# B&R Automation Studio project RobotNewEra
Automation Studio 4.2.4.149; 2.0.0

## Configuration APC820

CPU 5PC900.TS77-00, AutomationRuntime D4.21, Build 4.1.2, Safety 0.0

### Hardware
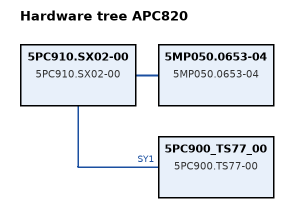
```
5MP050.0653-04 : 5MP050.0653-04 v1.0.3.0  [ETH1 -> 5PC910.SX02-00.IF3 (NodeNumber=1)]
  Terminal = true
  VncVcObjectName = Visu
  VncKeyMappingFile = VC\5MP050.0653-04.dis
  VncMaxConnections = 4
  VncRefreshRate = 100
5PC900_TS77_00 : 5PC900.TS77-00 v1.0.0.2  [SY -> 5PC910.SX02-00.SY1]
  UserRamDevice = APC8xx.SRAM
  UserRamSize = 770048
  RemMemDevice = APC8xx.SRAM
  RemMemSize = 261888
  PermanentPvSize = 10000
  RemanentGlobalPvSize = 81920
  VolatileGlobalPvSize = 500000
  PreservePermanentPvMemory = 1
  EnableUsbRemoteInstall = 1
  Connections = 8
  TimerDeviceType = EPLX2X
  TimerDevice = 5PC820.SX01-00.IF6
  TaskClassIdleTime = 8000
  Cyclic1Duration = 2000
  Cyclic1Tolerance = 0
  Cyclic1Stack = 40000
  Cyclic1Output = 1
  Cyclic2Duration = 30000
  Cyclic2Tolerance = 60000
  Cyclic2Stack = 28192
  Cyclic3Duration = 50000
  Cyclic3Tolerance = 200000
  Cyclic3Stack = 10240
  Cyclic4Duration = 100000
  Cyclic4Tolerance = 100000
  Cyclic5Duration = 200000
  Cyclic5Tolerance = 200000
  Cyclic6Duration = 500000
  Cyclic6Tolerance = 500000
  Cyclic7Duration = 1000000
  Cyclic7Tolerance = 1000000
  Cyclic8Duration = 30000
  Cyclic8Tolerance = 30000000
  Cyclic8Stack = 38192
5PC910.SX02-00 : 5PC910.SX02-00 v1.3.0.0
  Connector IF3:
    ActivateDevice = 1
    Mode = Manual
    InternetAddress = 192.168.1.9
    SubnetMask = 255.255.255.0
  Connector IF4:
    ActivateDevice = 1
    Mode = Manual
    SubnetMask = 255.255.255.0
```

### Cpu.per - 5PC900_TS77_00/Cpu.per
```iecst
(********************************************************************
 * COPYRIGHT --
 ********************************************************************
 * File: Cpu.per
 * Author: renj
 * Created: November 07, 2014
 ********************************************************************
 * Declaration of permanent variables
 ********************************************************************)
VAR_CONFIG
	HmiRetain AT %M0; (* *)
END_VAR
```

### AXESMap.ncm - 5PC900_TS77_00/Motion/AXESMap.ncm
```
NcMapping (NcSwId=ACP10)
  NcObject gAxisX (ModuleAddress=SDC_IF1.ST1, InterfaceType=SDC, Type=ncAXIS, Channel=1, AcoposSimulation=Off, InitParameter=sdc_i, AcoposParameter=sdc_p, AdditionalData=CNC_Enabled="1", Disabled=FALSE, ModuleDisabled=FALSE)
  NcObject gAxisY (ModuleAddress=SDC_IF1.ST2, InterfaceType=SDC, Type=ncAXIS, Channel=1, AcoposSimulation=Off, InitParameter=sdc_i, AcoposParameter=sdc_p, AdditionalData=CNC_Enabled="1", Disabled=FALSE)
  NcObject gAxisZ (ModuleAddress=SDC_IF1.ST3, InterfaceType=SDC, Type=ncAXIS, Channel=1, AcoposSimulation=Off, InitParameter=sdc_i, AcoposParameter=sdc_p, AdditionalData=CNC_Enabled="1", Disabled=FALSE)
  NcObject gAxisA (ModuleAddress=SDC_IF1.ST4, InterfaceType=SDC, Type=ncAXIS, Channel=1, AcoposSimulation=Off, InitParameter=sdc_i, AcoposParameter=sdc_p, AdditionalData=CNC_Enabled="1", Disabled=FALSE)
  NcObject gAxisB (ModuleAddress=SDC_IF1.ST5, InterfaceType=SDC, Type=ncAXIS, Channel=1, AcoposSimulation=Off, InitParameter=sdc_i, AcoposParameter=sdc_p, AdditionalData=CNC_Enabled="1", Disabled=FALSE)
  NcObject gAxisC (ModuleAddress=SDC_IF1.ST6, InterfaceType=SDC, Type=ncAXIS, Channel=1, AcoposSimulation=Off, InitParameter=sdc_i, AcoposParameter=sdc_p, AdditionalData=CNC_Enabled="1", Disabled=FALSE)
```

### Acp10cfg.ncc - 5PC900_TS77_00/Motion/Acp10cfg.ncc
```
NcConfiguration (Version=2.46.0, NcSwId=Acp10)
  ACP10CF1_typ:
    cnt_nettrc_rec_drive = 150
    bufsize_trace_upload = 1200
    tc_nc_man_task = Cyclic #1
    glob_pv_as_ncobject = Yes
    ncsys_dl_broadcast = Yes
    ncsys_dl_acp_reset = Yes
    safemc_log_err_to_ax = Yes
    network_init:
      ncsw_init_execute = Yes
      automatic_execute = No
      node_nr_warning = Yes
      net_err_before_ncact = Yes
    nettrc:
      enter_parsecrec = Yes
      enter_ncaction = Yes
      save_ring_startidx = No
    cam_prof_download:
      cam_dat_dl_parallel = No
      tc_cam_dl_parallel = Task class for NC Manager task
    plk_if[0]:
      if_name = IF6
      tc_CycDat_PLCopen = Task class for NC Manager task
      mc_broadcast_extdat = No
    sdc_if[0]:
      if_name = SDC_IF1
      mc_broadcast_size = 800
      mc_broadcast_extdat = No
```

### CNCMap.ncm - 5PC900_TS77_00/Motion/CNCMap.ncm
```
NcMapping (NcSwId=ARNC0)
  NcObject gRobot (Type=ncCNCSYS, Channel=1, AcoposSimulation=Off, InitParameter=cnc_i, Disabled=FALSE, ModuleDisabled=FALSE)
```

### MotionPvMa.vvm - 5PC900_TS77_00/Motion/MotionPvMa.vvm
```iecst
(********************************************************************
 * COPYRIGHT -- Bernecker + Rainer
 ********************************************************************
 * File: MotionPvMap.vvm
 * Author: radaka
 * Created: June 29, 2009
 ********************************************************************
 * PV mapping file
 ********************************************************************)
VAR_CONFIG
	Config.Config.Output.Monitor.ConfigOk AT %Q.Axes.Axes[0].Input.Parameter.ConfigOk; (*Insert your comment here...*)
	Config.Config.Output.Monitor.ConfigOk AT %Q.Cnc.Cnc[0].Input.Parameter.ConfigOk; (*Insert your comment here...*)
	Config.Config.Output.Monitor.ConfigOk AT %Q.System.System[0].Input.Parameter.ConfigOk; (*Insert your comment here...*)
	System.System[0].Output.Monitor.SystemAddress AT %Q.Config.Config.Input.Parameter.SystemAddress; (*Insert your comment here...*)
	Cnc.Cnc[0].Output.Monitor.CncAddress AT %Q.Config.Config.Input.Parameter.CncAddress; (*Insert your comment here...*)
	Axes.Axes[0].Output.Monitor.AxesAddress AT %Q.Config.Config.Input.Parameter.AxesAddress; (*Insert your comment here...*)
	Axes.Axes[0].Output.Monitor.AxesAddress AT %Q.System.System[0].Input.Parameter.AxesAddress; (*Insert your comment here...*)
	Cnc.Cnc[0].Output.Monitor.CncAddress AT %Q.System.System[0].Input.Parameter.CncAddress; (*Insert your comment here...*)
	Axes.Axes[0].Output.Monitor.AxesAddress AT %Q.Trf.AxesAddress; (*Only if TRF is used*)
	Cnc.Cnc[0].Output.Monitor.CncAddress AT %Q.Jog.CncAddress; (*Insert your comment here...*)
	Axes.Axes[0].Output.Monitor.AxesAddress AT %Q.6axATrqFF.AxesAddress; (*Insert your comment here...*)
END_VAR
```

## Configuration APC910

CPU 5PC900.TS77-02, AutomationRuntime N4.06, Build 4.1.2

### Task classes (Cpu.sw)
```

```

### Hardware
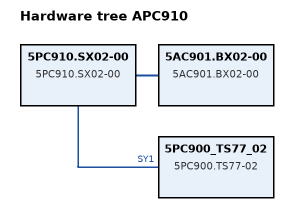
```
5AC901.BX02-00 : 5AC901.BX02-00 v1.0.0.2  [SY -> 5PC910.SX02-00.SY3]
5PC900_TS77_02 : 5PC900.TS77-02 v1.0.0.2  [SY -> 5PC910.SX02-00.SY1]
  Cyclic1Duration = 10000
  Cyclic1Tolerance = 10000
  Cyclic2Duration = 20000
  Cyclic2Tolerance = 20000
  Cyclic3Duration = 50000
  Cyclic3Tolerance = 50000
  Cyclic4Duration = 100000
  Cyclic4Tolerance = 100000
  Cyclic5Duration = 200000
  Cyclic5Tolerance = 200000
  Cyclic6Duration = 500000
  Cyclic6Tolerance = 500000
  Cyclic7Duration = 1000000
  Cyclic7Tolerance = 1000000
  Cyclic8Duration = 10000
  Cyclic8Tolerance = 30000000
5PC910.SX02-00 : 5PC910.SX02-00 v1.3.0.0
  Connector IF3:
    ActivateDevice = 1
    Mode = Manual
    InternetAddress = 192.168.0.9
    SubnetMask = 255.255.255.0
  Connector IF4:
    ActivateDevice = 1
    Mode = Manual
    InternetAddress = 192.168.1.9
    SubnetMask = 255.255.255.0
```

## Configuration Simulation

CPU , AutomationRuntime D4.24, Build 4.1.2, Safety 1.5

### Task classes (Cpu.sw)
```
Cyclic#1 (cycle 2000 us, tolerance 0 us):
  OptMotion <- MotionHandling.Optimizer.OptMotion.prg
  Cnc <- MotionHandling.CncHandling.Cnc.prg
  System <- MotionHandling.SystemHandling.System.prg (Version=1.00.1)
  Axes <- MotionHandling.AxesHandling.Axes.prg
  Jog <- MotionHandling.Jogging.Jog.prg
  Config <- MotionHandling.Configuration.Config.prg
  Trf <- MotionHandling.Transformations.Trf.prg
  myRecipe <- (binary)
Cyclic#2 (cycle 30000 us, tolerance 1200000 us):
  Error <- ErrorHandling.Error.prg  // Error Handling
  HmiKeyCtrl <- HmiHandling.HmiKeyCtrl.HmiKeyCtrl.prg
Cyclic#3 (cycle 20000 us, tolerance 10000000 us):
  HmiPrg <- HmiHandling.HmiPrg.HmiPrg.prg  // C++ Implementation FileExplorer
Cyclic#8 (cycle 30000 us, tolerance 30000000 us):
  HmiAlarm <- HmiHandling.HmiAlarm.HmiAlarm.prg
  HmiMain <- HmiHandling.HmiMain.HmiMain.prg
  HmiFile <- HmiHandling.HmiMain.HmiFile.prg
  HmiJogCtrl <- HmiHandling.HmiJog.HmiJogCtrl.prg
  RecipeCont <- Recipe.RecipeControl.prg
  UserStd <- UserStd.UserStd.prg  // User Management
  HmiHardKey <- HmiHandling.HmiHardKey.HmiHardKeyCtrl.prg  // HardKey Simulation
  HmiEditor <- HmiHandling.HmiEditor.HmiEditor.prg
  HmiFileVar <- HmiHandling.HmiEditor.HmiFileVar.prg
  HmiSetup <- HmiHandling.HmiSetup.HmiSetup.prg
NcDataObjects: sdc_p <- MotionHandling.MotionInitFiles.SDC.sdc_p.dob, ps_p <- MotionHandling.MotionInitFiles.ps_p.dob, sdc_i <- MotionHandling.MotionInitFiles.SDC.sdc_i.dob, AcpError <- MotionHandling.AxesHandling.AcpError.dob, sdc_j1_i <- MotionHandling.MotionInitFiles.SDC.sdc_j1_i.dob, sdc_j2_i <- MotionHandling.MotionInitFiles.SDC.sdc_j2_i.dob, sdc_j3_i <- MotionHandling.MotionInitFiles.SDC.sdc_j3_i.dob, sdc_j4_i <- MotionHandling.MotionInitFiles.SDC.sdc_j4_i.dob, JogInit <- MotionHandling.Jogging.JogInit.dob, sdc_j5_i <- MotionHandling.MotionInitFiles.SDC.sdc_j5_i.dob, sdc_j6_i <- MotionHandling.MotionInitFiles.SDC.sdc_j6_i.dob, JogPrg <- MotionHandling.Jogging.JogPrg.dob, robot_i <- MotionHandling.MotionInitFiles.robot_i.dob, gmcipsys <- MotionHandling.Interpreter.GmcIpConfig.gmcipsys.dob, gmciplbr <- MotionHandling.Interpreter.GmcIpConfig.gmciplbr.dob, gmcipcbr <- MotionHandling.Interpreter.GmcIpConfig.gmcipcbr.dob, gmciplsm <- MotionHandling.Interpreter.GmcIpConfig.gmciplsm.dob, gmcipcsm <- MotionHandling.Interpreter.GmcIpConfig.gmcipcsm.dob, gmcipcfg <- MotionHandling.Interpreter.GmcIpConfig.gmcipcfg.dob, gmcipiec <- MotionHandling.Interpreter.GmcIpConfig.gmcipiec.dob, gmciplog <- MotionHandling.Interpreter.GmcIpConfig.gmciplog.dob, gmcipesm <- MotionHandling.Interpreter.GmcIpConfig.gmcipesm.dob, gmcipmxd <- MotionHandling.Interpreter.GmcIpConfig.gmcipmxd.dob, gmcipmx <- MotionHandling.Interpreter.GmcIpConfig.gmcipmx.dob, gmcipvar <- MotionHandling.Interpreter.GmcIpUserConfig.gmcipvar.dob, gmcipfun <- MotionHandling.Interpreter.GmcIpUserConfig.gmcipfun.dob, gmcipfub <- MotionHandling.Interpreter.GmcIpUserConfig.gmcipfub.dob, gmcipubr <- MotionHandling.Interpreter.GmcIpUserConfig.gmcipubr.dob, gmcipusm <- MotionHandling.Interpreter.GmcIpUserConfig.gmcipusm.dob, gmcipus <- MotionHandling.Interpreter.GmcIpUserConfig.gmcipus.dob, gmcipuc <- MotionHandling.Interpreter.GmcIpUserConfig.gmcipuc.dob, TRFk_A1, gmcipvar1 <- GmcIpUserConfig.gmcipvar.dob, gmcipfun1 <- GmcIpUserConfig.gmcipfun.dob, gmcipfub1 <- GmcIpUserConfig.gmcipfub.dob, gmcipubr1 <- GmcIpUserConfig.gmcipubr.dob, gmcipusm1 <- GmcIpUserConfig.gmcipusm.dob, gmcipus1 <- GmcIpUserConfig.gmcipus.dob, gmcipuc1 <- GmcIpUserConfig.gmcipuc.dob, gmcipsys1 <- GmcIpConfig.gmcipsys.dob, gmciplbr1 <- GmcIpConfig.gmciplbr.dob, gmcipcbr1 <- GmcIpConfig.gmcipcbr.dob, gmciplsm1 <- GmcIpConfig.gmciplsm.dob, gmcipcsm1 <- GmcIpConfig.gmcipcsm.dob, gmcipcfg1 <- GmcIpConfig.gmcipcfg.dob, gmcipiec1 <- GmcIpConfig.gmcipiec.dob, gmciplog1 <- GmcIpConfig.gmciplog.dob, gmcipesm1 <- GmcIpConfig.gmcipesm.dob, gmcipmxd1 <- GmcIpConfig.gmcipmxd.dob, gmcipmx1 <- GmcIpConfig.gmcipmx.dob
VcDataObjects: MP50Ke <- Visualization.MP50Key.dob, Visu <- Visualization.Visu.dob
Binaries: arnc0001, TRFk_A0, Arnc0sys, sysconf, asfw, ashwd, arconfig, acp10cfg, arnc0map, arnc0cfg, acp10map, cncmap, axesmap, iomap, vcchtml, vccurl, vcxml, vcctrend, burgf5oe, vccpiech, arialgkb, vccbar, Vismp02, Vismp01, Vismp03, Visu203, Visu202, vcbclass, vccscale, MP50Ke01, vcpdsw, vcpfar00, vccdt, vccalarm, visvc, Visu01, vcdsloc, vcmgr, vctcal, arialbd, vcchspot, vccshape, vccpopup, vcnet, vcdsint, vcalarm, vccddbox, vccedit, courbd, vcfntttf, MP50Ke02, vccbmp, arialxsr, dejavz0z, vcclbox, vcctext, Visu03, vcrt, vccbtn, vccstr, vcgclass, arial, vccline, MP50Ke03, vcfile, vcshared, vccovl, Visu02, vcpdvnc, vccnum, vccslider
Libraries: Runtime, Operator, AsIecCon, astime, DataObj, AsMem, AsArLog, sys_lib, AsArProf, brsystem, FileIO, standard, asrfbext, AsICMP, AsUSB, visapi, AsIO, AsIOMMan, AsIODiag, AsSem, Acp10man, Acp10par, NcGlobal, Acp10_MC, Acp10sdc, Acp10sim, ModDiag, TRF_LIB, AsBrStr, powerlnk, MyLib, Arnc0ext, Arnc0man, Arnc0mx, loopconr, vcresman
```

### Hardware
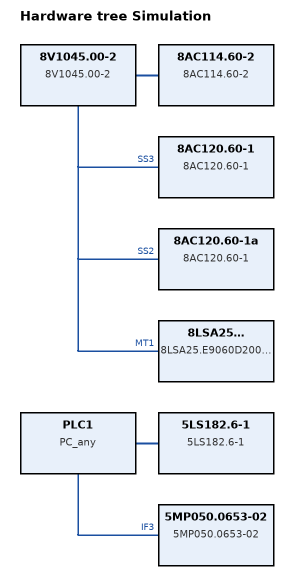
```
5LS182.6-1 : 5LS182.6-1 v1.2.6.0  [SL -> PLC1.SL1]
  Connector IF1:
    EplInterfaceRedundant = 0
    EplEthInterfaceRedundant = 0
5MP050.0653-02 : 5MP050.0653-02 v1.0.3.1  [ETH1 -> PLC1.IF3 (NodeNumber=1)]
  Terminal = true
  VncVcObjectName = Visu
  VncPortNumber = 5902
  VncMaxConnections = 8
  VncRefreshRate = 100
8AC114.60-2 : 8AC114.60-2 v1.0.0.8 (Disabled=true)  [SS -> 8V1045.00-2.SS1; PLK1 -> 5LS182.6-1.IF1 (NodeNumber=1)]
8AC120.60-1 : 8AC120.60-1 v1.0.0.2 (Disabled=true)  [SS -> 8V1045.00-2.SS3]
8AC120.60-1a : 8AC120.60-1 v1.0.0.2 (Disabled=true)  [SS -> 8V1045.00-2.SS2]
8LSA25.E9060D200-0 : 8LSA25.E9060D200-0 v1.0.1.34 (Disabled=true)  [MT -> 8V1045.00-2.MT1]
8V1045.00-2 : 8V1045.00-2 v1.0.0.2 (Disabled=true)
  CNC_r1 = on
PLC1 : PC_any v1.1.0.0 (OrderNumber=PC)
  Connector IF3:
    Vnc1
    VncVcObjectName1 = MP50Ke
    VncAuthentication1 = 1
    VncPasswordViewOnly1 = v
    VncPasswordViewControl1 = c
    VncPortNumber1 = 5901
    VncMaxConnections1 = 8
    VncRefreshRate1 = 500
  RemanentGlobalPvSize = 81920
  VolatileGlobalPvSize = 3000000
  PreserveNonVolatileSystemSettings = 0
  SystemTick = 2000
  TaskClassIdleTime = 4000
  XLinkUseDefault = 0
  XLinkDuration = 50000
  Cyclic1Duration = 2000
  Cyclic1Tolerance = 0
  Cyclic1Stack = 30000
  Cyclic1Output = 2
  Cyclic2Duration = 30000
  Cyclic2Tolerance = 1200000
  Cyclic3Duration = 20000
  Cyclic3Tolerance = 10000000
  Cyclic4Duration = 1006000
  Cyclic4Tolerance = 10060000
  Cyclic5Duration = 2006000
  Cyclic5Tolerance = 10030000
  Cyclic6Duration = 3000000
  Cyclic6Tolerance = 12000000
  Cyclic7Duration = 4006000
  Cyclic7Tolerance = 12018000
  Cyclic8Duration = 30000
  Cyclic8Tolerance = 30000000
  Cyclic8Stack = 28196
  FileDevice1
  FileDeviceName1 = CNC_PrgDir
  FileDevicePath1 = C:\Data\Programs
```

### Hmi.vvm - PLC1/HmiMap/Hmi.vvm
```iecst
(********************************************************************
 * COPYRIGHT --
 ********************************************************************
 * File: Hmi.vvm
 * Author: renj
 * Created: July 28, 2014
 ********************************************************************
 * PV mapping file
 ********************************************************************)
VAR_CONFIG
	::System:System[0].Output.Monitor.SystemAddress AT %Q.::HmiGlobal.Address.SystemAddress; (*Insert your comment here...*)
	::Cnc:Cnc[0].Output.Monitor.CncAddress AT %Q.::HmiGlobal.Address.CncAddress; (*Insert your comment here...*)
	::Axes:Axes[0].Output.Monitor.AxesAddress AT %Q.::HmiGlobal.Address.AxesAddress; (*Insert your comment here...*)
	::Jog:Jogging.JogAddress AT %Q.::HmiGlobal.Address.JogAddress; (*Insert your comment here...*)
	::RecipeCont:Recipe.Monitor.RecipeAddress AT %Q.::HmiGlobal.Address.RecipeAddress; (*Insert your comment here...*)
	::Error:Error.Output.Monitor.ErrorHandlingAddress AT %Q.::HmiGlobal.Address.ErrorAddress; (*Insert your comment here...*)
END_VAR
```

### AXESMap.ncm - PLC1/Motion/AXESMap.ncm
```
NcMapping (NcSwId=ACP10)
  NcObject gPowerSupply (ModuleAddress=SDC_IF1.ST7, InterfaceType=SDC, Type=ncAXIS, Channel=1, AcoposSimulation=Off, InitParameter=sdc_i, Disabled=FALSE)
  NcObject gAxisQ1 (ModuleAddress=SDC_IF1.ST8, InterfaceType=SDC, Type=ncAXIS, Channel=1, AcoposSimulation=Off, InitParameter=sdc_j1_i, AcoposParameter=sdc_p, AdditionalData=CNC_Enabled="1", Disabled=FALSE)
  NcObject gAxisQ2 (ModuleAddress=SDC_IF1.ST9, InterfaceType=SDC, Type=ncAXIS, Channel=1, AcoposSimulation=Off, InitParameter=sdc_j2_i, AcoposParameter=sdc_p, AdditionalData=CNC_Enabled="1", Disabled=FALSE)
  NcObject gAxisQ3 (ModuleAddress=SDC_IF1.ST10, InterfaceType=SDC, Type=ncAXIS, Channel=1, AcoposSimulation=Off, InitParameter=sdc_j3_i, AcoposParameter=sdc_p, AdditionalData=CNC_Enabled="1", Disabled=FALSE)
  NcObject gAxisQ4 (ModuleAddress=SDC_IF1.ST11, InterfaceType=SDC, Type=ncAXIS, Channel=1, AcoposSimulation=Off, InitParameter=sdc_j4_i, AcoposParameter=sdc_p, AdditionalData=CNC_Enabled="1", Disabled=FALSE)
  NcObject gAxisQ5 (ModuleAddress=SDC_IF1.ST12, InterfaceType=SDC, Type=ncAXIS, Channel=1, AcoposSimulation=Off, InitParameter=sdc_j5_i, AcoposParameter=sdc_p, AdditionalData=CNC_Enabled="1", Disabled=FALSE)
  NcObject gAxisQ6 (ModuleAddress=SDC_IF1.ST13, InterfaceType=SDC, Type=ncAXIS, Channel=1, AcoposSimulation=Off, InitParameter=sdc_j6_i, AcoposParameter=sdc_p, AdditionalData=CNC_Enabled="1", Disabled=FALSE)
  NcObject gAxisX (ModuleAddress=SDC_IF1.ST1, InterfaceType=SDC, Type=ncAXIS, Channel=1, AcoposSimulation=Off, InitParameter=sdc_i, AcoposParameter=sdc_p, AdditionalData=CNC_Enabled="1", Disabled=FALSE, ModuleDisabled=FALSE)
  NcObject gAxisY (ModuleAddress=SDC_IF1.ST2, InterfaceType=SDC, Type=ncAXIS, Channel=1, AcoposSimulation=Off, InitParameter=sdc_i, AcoposParameter=sdc_p, AdditionalData=CNC_Enabled="1", Disabled=FALSE)
  NcObject gAxisZ (ModuleAddress=SDC_IF1.ST3, InterfaceType=SDC, Type=ncAXIS, Channel=1, AcoposSimulation=Off, InitParameter=sdc_i, AcoposParameter=sdc_p, AdditionalData=CNC_Enabled="1", Disabled=FALSE)
  NcObject gAxisA (ModuleAddress=SDC_IF1.ST4, InterfaceType=SDC, Type=ncAXIS, Channel=1, AcoposSimulation=Off, InitParameter=sdc_i, AcoposParameter=sdc_p, AdditionalData=CNC_Enabled="1", Disabled=FALSE)
  NcObject gAxisB (ModuleAddress=SDC_IF1.ST5, InterfaceType=SDC, Type=ncAXIS, Channel=1, AcoposSimulation=Off, InitParameter=sdc_i, AcoposParameter=sdc_p, AdditionalData=CNC_Enabled="1", Disabled=FALSE)
  NcObject gAxisC (ModuleAddress=SDC_IF1.ST6, InterfaceType=SDC, Type=ncAXIS, Channel=1, AcoposSimulation=Off, InitParameter=sdc_i, AcoposParameter=sdc_p, AdditionalData=CNC_Enabled="1", Disabled=FALSE)
```

### Acp10cfg.ncc - PLC1/Motion/Acp10cfg.ncc
```
NcConfiguration (Version=2.43.0, NcSwId=Acp10)
  ACP10CF1_typ:
    cnt_nettrc_rec_drive = 1500
    bufsize_trace_upload = 1200
    tc_nc_man_task = Cyclic #1
    glob_pv_as_ncobject = Yes
    ncsys_dl_broadcast = Yes
    ncsys_dl_acp_reset = Yes
    safemc_log_err_to_ax = Yes
    network_init:
      ncsw_init_execute = Yes
      automatic_execute = No
      node_nr_warning = Yes
      net_err_before_ncact = Yes
    nettrc:
      enter_parsecrec = Yes
      enter_ncaction = Yes
      save_ring_startidx = Yes
    cam_prof_download:
      cam_dat_dl_parallel = No
      tc_cam_dl_parallel = Task class for NC Manager task
    plk_if[0]:
      if_name = SL1.IF1
      tc_CycDat_PLCopen = Task class for NC Manager task
      mc_broadcast_extdat = No
    sdc_if[0]:
      if_name = SDC_IF1
      mc_broadcast_size = 800
      mc_broadcast_extdat = No
```

### Acp10map.ncm - PLC1/Motion/Acp10map.ncm
```
NcMapping (NcSwId=Acp10)
  NcObject gPowerSupply (ModuleId=8B0Pxxxxxxxx.xxx-x, Type=ncAXIS, Channel=1, AcoposSimulation=Off, InitParameter=sdc_i, Disabled=TRUE, ModuleDisabled=FALSE)
  NcObject gAxisQ1 (ModuleId=8BVIxxxxxxDx.xxx-x, Type=ncAXIS, Channel=1, AcoposSimulation=Off, InitParameter=joint1_i, AcoposParameter=acpm_p, AdditionalData=CNC_Enabled="1", Disabled=TRUE, ModuleDisabled=FALSE)
  NcObject gAxisQ2 (ModuleId=8BVIxxxxxxDx.xxx-x, Type=ncAXIS, Channel=2, AcoposSimulation=Off, InitParameter=joint2_i, AcoposParameter=acpm_p, AdditionalData=CNC_Enabled="1", Disabled=TRUE, ModuleDisabled=FALSE)
  NcObject gAxisQ3 (ModuleId=8BVIxxxxxxDx.xxx-x1, Type=ncAXIS, Channel=1, AcoposSimulation=Off, InitParameter=joint3_i, AcoposParameter=acpm_p, AdditionalData=CNC_Enabled="1", Disabled=TRUE, ModuleDisabled=FALSE)
  NcObject gAxisQ4 (ModuleId=8BVIxxxxxxDx.xxx-x1, Type=ncAXIS, Channel=2, AcoposSimulation=Off, InitParameter=joint4_i, AcoposParameter=acpmic_p, AdditionalData=CNC_Enabled="1", Disabled=TRUE, ModuleDisabled=FALSE)
  NcObject gAxisQ5 (ModuleId=8BVIxxxxxxDx.xxx-x2, Type=ncAXIS, Channel=1, AcoposSimulation=Off, InitParameter=joint5_i, AcoposParameter=acpmic_p, AdditionalData=CNC_Enabled="1", Disabled=TRUE, ModuleDisabled=FALSE)
  NcObject gAxisQ6 (ModuleId=8BVIxxxxxxDx.xxx-x2, Type=ncAXIS, Channel=2, AcoposSimulation=Off, InitParameter=joint6_i, AcoposParameter=acpmic_p1, AdditionalData=CNC_Enabled="1", Disabled=TRUE, ModuleDisabled=FALSE)
  NcObject gAxis02 (ModuleId=8V1045.00-2, Type=ncAXIS, Channel=1, AcoposSimulation=Off, InitParameter=gAxis02i, AcoposParameter=gAxis02a, AdditionalData=CNC_Enabled="1" , Disabled=TRUE, ModuleDisabled=FALSE)
  NcObject 8V1045.00-2_ncV_AXIS1 (ModuleId=8V1045.00-2, Type=ncV_AXIS, Channel=1, Disabled=TRUE, ModuleDisabled=FALSE)
```

### Arnc0cfg.ncc - PLC1/Motion/Arnc0cfg.ncc
```
NcConfiguration (Version=1.38.0, NcSwId=arnc0)
  ARNC0CFG_typ:
    sampling_rate = 2000
    cnt_nettrc_rec_drive = 1500
    bufsize_sys_trace = 16#00005000
    enable_mp_log = Yes
    tc_nc_man_task = Cyclic #1
    bg_load = 1
    glob_pv_as_ncobject = Yes
```

### CNCMap.ncm - PLC1/Motion/CNCMap.ncm
```
NcMapping (NcSwId=ARNC0, DisabledNodesAreHidden=False)
  NcObject gRobot (Type=ncCNCSYS, Channel=1, AcoposSimulation=Off, InitParameter=robot_i, Disabled=FALSE, ModuleDisabled=FALSE)
```

### MotionPvMa.vvm - PLC1/Motion/MotionPvMa.vvm
```iecst
(********************************************************************
 * COPYRIGHT -- Bernecker + Rainer
 ********************************************************************
 * File: MotionPvMap.vvm
 * Author: radaka
 * Created: June 29, 2009
 ********************************************************************
 * PV mapping file
 ********************************************************************)
VAR_CONFIG
	Config.Config.Output.Monitor.ConfigOk AT %Q.Axes.Axes[0].Input.Parameter.ConfigOk; (*Insert your comment here...*)
	Config.Config.Output.Monitor.ConfigOk AT %Q.Cnc.Cnc[0].Input.Parameter.ConfigOk; (*Insert your comment here...*)
	Config.Config.Output.Monitor.ConfigOk AT %Q.System.System[0].Input.Parameter.ConfigOk; (*Insert your comment here...*)
	System.System[0].Output.Monitor.SystemAddress AT %Q.Config.Config.Input.Parameter.SystemAddress; (*Insert your comment here...*)
	Cnc.Cnc[0].Output.Monitor.CncAddress AT %Q.Config.Config.Input.Parameter.CncAddress; (*Insert your comment here...*)
	Axes.Axes[0].Output.Monitor.AxesAddress AT %Q.Config.Config.Input.Parameter.AxesAddress; (*Insert your comment here...*)
	Axes.Axes[0].Output.Monitor.AxesAddress AT %Q.System.System[0].Input.Parameter.AxesAddress; (*Insert your comment here...*)
	Cnc.Cnc[0].Output.Monitor.CncAddress AT %Q.System.System[0].Input.Parameter.CncAddress; (*Insert your comment here...*)
	Axes.Axes[0].Output.Monitor.AxesAddress AT %Q.Trf.AxesAddress; (*Only if TRF is used*)
	Cnc.Cnc[0].Output.Monitor.CncAddress AT %Q.Jog.CncAddress; (*Insert your comment here...*)
END_VAR
```

## Configuration X20CP1486

CPU X20CP1486, AutomationRuntime S3.09, Build 4.1.2

### Task classes (Cpu.sw)
```
Cyclic#1 (cycle 2000 us, tolerance 0 us):
  6axATrqFF <- MotionHandling.FeedForward.6axATrqFF.prg
  Config <- MotionHandling.Configuration.Config.prg
  System <- MotionHandling.SystemHandling.System.prg
  Cnc <- MotionHandling.CncHandling.Cnc.prg
  Axes <- MotionHandling.AxesHandling.Axes.prg
  OptMotion <- MotionHandling.Optimizer.OptMotion.prg
  Jog <- MotionHandling.Jogging.Jog.prg
  Trf <- MotionHandling.Transformations.Trf.prg
Cyclic#2 (cycle 30000 us, tolerance 30000 us):
  Error <- ErrorHandling.Error.prg
  HmiKeyCtrl <- HmiHandling.HmiKeyCtrl.HmiKeyCtrl.prg
  HmiHardKey <- HmiHandling.HmiHardKey.HmiHardKeyCtrl.prg
Cyclic#3 (cycle 20000 us, tolerance 40000 us):
  HmiPrg <- HmiHandling.HmiPrg.HmiPrg.prg
Cyclic#8 (cycle 30000 us, tolerance 30000000 us):
  HmiAlarm <- HmiHandling.HmiAlarm.HmiAlarm.prg
  HmiMain <- HmiHandling.HmiMain.HmiMain.prg
  HmiFile <- HmiHandling.HmiMain.HmiFile.prg
  HmiJogCtrl <- HmiHandling.HmiJog.HmiJogCtrl.prg
  RecipeCont <- Recipe.RecipeControl.prg
  UserStd <- UserStd.UserStd.prg
  HmiEditor <- HmiHandling.HmiEditor.HmiEditor.prg
  HmiFileVar <- HmiHandling.HmiEditor.HmiFileVar.prg
  HmiSetup <- HmiHandling.HmiSetup.HmiSetup.prg
NcDataObjects: sdc_i <- MotionHandling.MotionInitFiles.SDC.sdc_i.dob, sdc_p <- MotionHandling.MotionInitFiles.SDC.sdc_p.dob, ps_p <- MotionHandling.MotionInitFiles.ps_p.dob, acpm_p <- MotionHandling.MotionInitFiles.acpm_p.dob, acpmic_p <- MotionHandling.MotionInitFiles.acpmic_p.dob, joint1_i <- MotionHandling.MotionInitFiles.joint1_i.dob, joint2_i <- MotionHandling.MotionInitFiles.joint2_i.dob, joint3_i <- MotionHandling.MotionInitFiles.joint3_i.dob, joint4_i <- MotionHandling.MotionInitFiles.joint4_i.dob, joint5_i <- MotionHandling.MotionInitFiles.joint5_i.dob, joint6_i <- MotionHandling.MotionInitFiles.joint6_i.dob, AcpError <- MotionHandling.AxesHandling.AcpError.dob, JogInit <- MotionHandling.Jogging.JogInit.dob, JogPrg <- MotionHandling.Jogging.JogPrg.dob, robot_i <- MotionHandling.MotionInitFiles.robot_i.dob, gmcipsys <- MotionHandling.Interpreter.GmcIpConfig.gmcipsys.dob, gmciplbr <- MotionHandling.Interpreter.GmcIpConfig.gmciplbr.dob, gmcipcbr <- MotionHandling.Interpreter.GmcIpConfig.gmcipcbr.dob, gmciplsm <- MotionHandling.Interpreter.GmcIpConfig.gmciplsm.dob, gmcipcsm <- MotionHandling.Interpreter.GmcIpConfig.gmcipcsm.dob, gmcipcfg <- MotionHandling.Interpreter.GmcIpConfig.gmcipcfg.dob, gmcipiec <- MotionHandling.Interpreter.GmcIpConfig.gmcipiec.dob, gmciplog <- MotionHandling.Interpreter.GmcIpConfig.gmciplog.dob, gmcipesm <- MotionHandling.Interpreter.GmcIpConfig.gmcipesm.dob, gmcipmxd <- MotionHandling.Interpreter.GmcIpConfig.gmcipmxd.dob, gmcipmx <- MotionHandling.Interpreter.GmcIpConfig.gmcipmx.dob, gmcipvar <- MotionHandling.Interpreter.GmcIpUserConfig.gmcipvar.dob, gmcipfun <- MotionHandling.Interpreter.GmcIpUserConfig.gmcipfun.dob, gmcipfub <- MotionHandling.Interpreter.GmcIpUserConfig.gmcipfub.dob, gmcipubr <- MotionHandling.Interpreter.GmcIpUserConfig.gmcipubr.dob, gmcipusm <- MotionHandling.Interpreter.GmcIpUserConfig.gmcipusm.dob, gmcipus <- MotionHandling.Interpreter.GmcIpUserConfig.gmcipus.dob, gmcipuc <- MotionHandling.Interpreter.GmcIpUserConfig.gmcipuc.dob
Binaries: vccedit, vccscale, dejavz0z, arialxsr, vccslider, vccalarm, vccpopup, vccline, vccstr, courbd, Visu03, vccddbox, vccshape, Visu02, Visu01, vccdt, vcclbox, vcpkat, vcfntttf, vccbmp, vcshared, vcmgr, vcfile, vcgclass, arial, vcchspot, vcdsint, vccbtn, vcdsloc, vccovl, vcpfx20, vcctext, vcalarm, vcbclass, visvc, vcrt, vccnum, arialbd, vcpdsw, vcnet, vcpdvnc, vctcal, ashwd, arconfig, asfw, sysconf, iomap, Arnc0map, Arnc0Map1, Acp10Map1, arnc0cfg, acp10cfg, Acp10map, Acp10sys, Arnc0sys, MP50Ke01, MP50Ke03, MP50Ke02
Libraries: Runtime, Operator, AsIecCon, astime, DataObj, AsMem, AsArLog, sys_lib, AsArProf, brsystem, FileIO, standard, asrfbext, AsICMP, AsUSB, visapi, TRF_LIB, AsIO, AsIOMMan, AsIODiag, AsSem, AsBrStr, Arnc0ext, MyLib, LoopConR, Acp10man, Acp10par, NcGlobal, Arnc0man, Acp10sdc, Acp10sim, Acp10_MC, Arnc0mx, powerlnk, ModDiag, vcresman, ashw
```

### Hardware
```
X20CP1486 : X20CP1486 v1.1.4.0
  Connector IF2:
    ActivateDevice = 1
  Connector IF3:
    EplEthInterfaceRedundant = 0
  RemanentGlobalPvSize = 81920
  VolatileGlobalPvSize = 3000000
  PreserveNonVolatileSystemSettings = 0
  SystemTick = 2000
  TaskClassIdleTime = 4000
  Cyclic1Duration = 2000
  Cyclic1Tolerance = 0
  Cyclic1Stack = 30000
  Cyclic1Output = 1
  Cyclic2Duration = 30000
  Cyclic2Tolerance = 30000
  Cyclic3Duration = 20000
  Cyclic3Tolerance = 40000
  Cyclic4Duration = 100000
  Cyclic4Tolerance = 100000
  Cyclic5Duration = 200000
  Cyclic5Tolerance = 200000
  Cyclic6Duration = 500000
  Cyclic6Tolerance = 500000
  Cyclic7Duration = 1000000
  Cyclic7Tolerance = 1000000
  Cyclic8Duration = 30000
  Cyclic8Tolerance = 30000000
  Cyclic8Stack = 28196
  FileDevice1
  FileDeviceName1 = CNC_PrgDir
  FileDevicePath1 = C:\Data\Programs
  EthernetHostName = luxiaochun
```

### Acp10Map1.ncm - X20CP1486/Motion/Acp10Map1.ncm
```
NcMapping (NcSwId=ACP10, DisabledNodesAreHidden=False)
  NcObject gPowerSupply (ModuleAddress=SDC_IF1.ST7, InterfaceType=SDC, Type=ncAXIS, Channel=1, AcoposSimulation=Off, InitParameter=sdc_i, Disabled=FALSE)
  NcObject gAxisQ1 (ModuleAddress=SDC_IF1.ST8, InterfaceType=SDC, Type=ncAXIS, Channel=1, AcoposSimulation=Off, InitParameter=sdc_j1_i, AcoposParameter=sdc_p, AdditionalData=CNC_Enabled="1", Disabled=FALSE)
  NcObject gAxisQ2 (ModuleAddress=SDC_IF1.ST9, InterfaceType=SDC, Type=ncAXIS, Channel=1, AcoposSimulation=Off, InitParameter=sdc_j2_i, AcoposParameter=sdc_p, AdditionalData=CNC_Enabled="1", Disabled=FALSE)
  NcObject gAxisQ3 (ModuleAddress=SDC_IF1.ST10, InterfaceType=SDC, Type=ncAXIS, Channel=1, AcoposSimulation=Off, InitParameter=sdc_j3_i, AcoposParameter=sdc_p, AdditionalData=CNC_Enabled="1", Disabled=FALSE)
  NcObject gAxisQ4 (ModuleAddress=SDC_IF1.ST11, InterfaceType=SDC, Type=ncAXIS, Channel=1, AcoposSimulation=Off, InitParameter=sdc_j4_i, AcoposParameter=sdc_p, AdditionalData=CNC_Enabled="1", Disabled=FALSE)
  NcObject gAxisQ5 (ModuleAddress=SDC_IF1.ST12, InterfaceType=SDC, Type=ncAXIS, Channel=1, AcoposSimulation=Off, InitParameter=sdc_j5_i, AcoposParameter=sdc_p, AdditionalData=CNC_Enabled="1", Disabled=FALSE)
  NcObject gAxisQ6 (ModuleAddress=SDC_IF1.ST13, InterfaceType=SDC, Type=ncAXIS, Channel=1, AcoposSimulation=Off, InitParameter=sdc_j6_i, AcoposParameter=sdc_p, AdditionalData=CNC_Enabled="1", Disabled=FALSE)
  NcObject gAxisX (ModuleAddress=SDC_IF1.ST1, InterfaceType=SDC, Type=ncAXIS, Channel=1, AcoposSimulation=Off, InitParameter=sdc_i, AcoposParameter=sdc_p, AdditionalData=CNC_Enabled="1", Disabled=FALSE)
  NcObject gAxisY (ModuleAddress=SDC_IF1.ST2, InterfaceType=SDC, Type=ncAXIS, Channel=1, AcoposSimulation=Off, InitParameter=sdc_i, AcoposParameter=sdc_p, AdditionalData=CNC_Enabled="1", Disabled=FALSE)
  NcObject gAxisZ (ModuleAddress=SDC_IF1.ST3, InterfaceType=SDC, Type=ncAXIS, Channel=1, AcoposSimulation=Off, InitParameter=sdc_i, AcoposParameter=sdc_p, AdditionalData=CNC_Enabled="1", Disabled=FALSE)
  NcObject gAxisA (ModuleAddress=SDC_IF1.ST4, InterfaceType=SDC, Type=ncAXIS, Channel=1, AcoposSimulation=Off, InitParameter=sdc_i, AcoposParameter=sdc_p, AdditionalData=CNC_Enabled="1", Disabled=FALSE)
  NcObject gAxisB (ModuleAddress=SDC_IF1.ST5, InterfaceType=SDC, Type=ncAXIS, Channel=1, AcoposSimulation=Off, InitParameter=sdc_i, AcoposParameter=sdc_p, AdditionalData=CNC_Enabled="1", Disabled=FALSE)
  NcObject gAxisC (ModuleAddress=SDC_IF1.ST6, InterfaceType=SDC, Type=ncAXIS, Channel=1, AcoposSimulation=Off, InitParameter=sdc_i, AcoposParameter=sdc_p, AdditionalData=CNC_Enabled="1", Disabled=FALSE)
```

### Acp10cfg.ncc - X20CP1486/Motion/Acp10cfg.ncc
```
NcConfiguration (Version=2.47.2, NcSwId=Acp10)
  ACP10CF1_typ:
    cnt_nettrc_rec_drive = 1500
    bufsize_trace_upload = 1200
    tc_nc_man_task = Cyclic #1
    glob_pv_as_ncobject = Yes
    ncsys_dl_broadcast = Yes
    ncsys_dl_acp_reset = Yes
    safemc_log_err_to_ax = Yes
    network_init:
      ncsw_init_execute = Yes
      automatic_execute = No
      node_nr_warning = Yes
      net_err_before_ncact = Yes
    nettrc:
      enter_parsecrec = Yes
      enter_ncaction = Yes
      save_ring_startidx = Yes
    cam_prof_download:
      cam_dat_dl_parallel = No
      tc_cam_dl_parallel = Task class for NC Manager task
    sdc_if[0]:
      if_name = SDC_IF1
      mc_broadcast_size = 800
      mc_broadcast_extdat = No
```

### Arnc0Map1.ncm - X20CP1486/Motion/Arnc0Map1.ncm
```
NcMapping (NcSwId=ARNC0, DisabledNodesAreHidden=False)
  NcObject gRobot (Type=ncCNCSYS, Channel=1, AcoposSimulation=Off, InitParameter=robot_i, Disabled=FALSE)
```

### Arnc0cfg.ncc - X20CP1486/Motion/Arnc0cfg.ncc
```
NcConfiguration (Version=2.47.4, NcSwId=Arnc0)
  ARNC0CFG_typ:
    sampling_rate = 2000
    cnt_nettrc_rec_drive = 1500
    bufsize_sys_trace = 16#00005000
    enable_mp_log = Yes
    tc_nc_man_task = Cyclic #1
    bg_load = 1
    glob_pv_as_ncobject = Yes
```

### MotionPvMa.vvm - X20CP1486/Motion/MotionPvMa.vvm
```iecst
(********************************************************************
 * COPYRIGHT -- Bernecker + Rainer
 ********************************************************************
 * File: MotionPvMap.vvm
 * Author: radaka
 * Created: June 29, 2009
 ********************************************************************
 * PV mapping file
 ********************************************************************)
VAR_CONFIG
	::Config:Config.Output.Monitor.ConfigOk AT %Q.::Axes:Axes[0].Input.Parameter.ConfigOk; (*Insert your comment here...*)
	::Config:Config.Output.Monitor.ConfigOk AT %Q.::Cnc:Cnc[0].Input.Parameter.ConfigOk; (*Insert your comment here...*)
	::Config:Config.Output.Monitor.ConfigOk AT %Q.::System:System[0].Input.Parameter.ConfigOk; (*Insert your comment here...*)
	::System:System[0].Output.Monitor.SystemAddress AT %Q.::Config:Config.Input.Parameter.SystemAddress; (*Insert your comment here...*)
	::Cnc:Cnc[0].Output.Monitor.CncAddress AT %Q.::Config:Config.Input.Parameter.CncAddress; (*Insert your comment here...*)
	::Axes:Axes[0].Output.Monitor.AxesAddress AT %Q.::Config:Config.Input.Parameter.AxesAddress; (*Insert your comment here...*)
	::Axes:Axes[0].Output.Monitor.AxesAddress AT %Q.::System:System[0].Input.Parameter.AxesAddress; (*Insert your comment here...*)
	::Cnc:Cnc[0].Output.Monitor.CncAddress AT %Q.::System:System[0].Input.Parameter.CncAddress; (*Insert your comment here...*)
	::Axes:Axes[0].Output.Monitor.AxesAddress AT %Q.::Trf:AxesAddress; (*Only if TRF is used*)
	::Cnc:Cnc[0].Output.Monitor.CncAddress AT %Q.::Jog:CncAddress; (*Insert your comment here...*)
END_VAR
```

## Configuration X20CP1586

CPU , AutomationRuntime G4.06, Build 4.1.2, Safety 0.0

### Task classes (Cpu.sw)
```
Cyclic#1 (cycle 4000 us, tolerance 0 us):
  6axATrqFF <- MotionHandling.FeedForward.6axATrqFF.prg
  OptMotion <- MotionHandling.Optimizer.OptMotion.prg
  Config <- MotionHandling.Configuration.Config.prg
  System <- MotionHandling.SystemHandling.System.prg
  Cnc <- MotionHandling.CncHandling.Cnc.prg
  Axes <- MotionHandling.AxesHandling.Axes.prg
  Jog <- MotionHandling.Jogging.Jog.prg
  Trf <- MotionHandling.Transformations.Trf.prg
Cyclic#2 (cycle 30000 us, tolerance 30000 us):
  Error <- ErrorHandling.Error.prg
  HmiKeyCtrl <- HmiHandling.HmiKeyCtrl.HmiKeyCtrl.prg
  HmiHardKey <- HmiHandling.HmiHardKey.HmiHardKeyCtrl.prg
Cyclic#3 (cycle 20000 us, tolerance 30000000 us):
  HmiPrg <- HmiHandling.HmiPrg.HmiPrg.prg
Cyclic#8 (cycle 30000 us, tolerance 30000000 us):
  HmiAlarm <- HmiHandling.HmiAlarm.HmiAlarm.prg
  HmiMain <- HmiHandling.HmiMain.HmiMain.prg
  HmiFile <- HmiHandling.HmiMain.HmiFile.prg
  HmiJogCtrl <- HmiHandling.HmiJog.HmiJogCtrl.prg
  HmiEditor <- HmiHandling.HmiEditor.HmiEditor.prg
  HmiFileVar <- HmiHandling.HmiEditor.HmiFileVar.prg
  RecipeCont <- Recipe.RecipeControl.prg
  HmiSetup <- HmiHandling.HmiSetup.HmiSetup.prg
  UserStd <- UserStd.UserStd.prg
  HmiIO <- HmiHandling.HmiIO.HmiIO.prg [disabled]
DataObjects: Acp10sys, Arnc0sys
NcDataObjects: sdc_i <- MotionHandling.MotionInitFiles.SDC.sdc_i.dob, sdc_p <- MotionHandling.MotionInitFiles.SDC.sdc_p.dob, ps_p <- MotionHandling.MotionInitFiles.ps_p.dob, acpm_p <- MotionHandling.MotionInitFiles.acpm_p.dob, acpmic_p <- MotionHandling.MotionInitFiles.acpmic_p.dob, sdc_j1_i <- MotionHandling.MotionInitFiles.SDC.sdc_j1_i.dob, sdc_j2_i <- MotionHandling.MotionInitFiles.SDC.sdc_j2_i.dob, sdc_j3_i <- MotionHandling.MotionInitFiles.SDC.sdc_j3_i.dob, sdc_j4_i <- MotionHandling.MotionInitFiles.SDC.sdc_j4_i.dob, sdc_j5_i <- MotionHandling.MotionInitFiles.SDC.sdc_j5_i.dob, sdc_j6_i <- MotionHandling.MotionInitFiles.SDC.sdc_j6_i.dob, JogInit <- MotionHandling.Jogging.JogInit.dob, JogPrg <- MotionHandling.Jogging.JogPrg.dob, robot_i <- MotionHandling.MotionInitFiles.robot_i.dob, AcpError <- MotionHandling.AxesHandling.AcpError.dob, gmcipsys <- MotionHandling.Interpreter.GmcIpConfig.gmcipsys.dob, gmciplbr <- MotionHandling.Interpreter.GmcIpConfig.gmciplbr.dob, gmcipcbr <- MotionHandling.Interpreter.GmcIpConfig.gmcipcbr.dob, gmciplsm <- MotionHandling.Interpreter.GmcIpConfig.gmciplsm.dob, gmcipcsm <- MotionHandling.Interpreter.GmcIpConfig.gmcipcsm.dob, gmcipcfg <- MotionHandling.Interpreter.GmcIpConfig.gmcipcfg.dob, gmcipiec <- MotionHandling.Interpreter.GmcIpConfig.gmcipiec.dob, gmciplog <- MotionHandling.Interpreter.GmcIpConfig.gmciplog.dob, gmcipesm <- MotionHandling.Interpreter.GmcIpConfig.gmcipesm.dob, gmcipmxd <- MotionHandling.Interpreter.GmcIpConfig.gmcipmxd.dob, gmcipmx <- MotionHandling.Interpreter.GmcIpConfig.gmcipmx.dob, gmcipvar <- MotionHandling.Interpreter.GmcIpUserConfig.gmcipvar.dob, gmcipfun <- MotionHandling.Interpreter.GmcIpUserConfig.gmcipfun.dob, gmcipfub <- MotionHandling.Interpreter.GmcIpUserConfig.gmcipfub.dob, gmcipubr <- MotionHandling.Interpreter.GmcIpUserConfig.gmcipubr.dob, gmcipusm <- MotionHandling.Interpreter.GmcIpUserConfig.gmcipusm.dob, gmcipus <- MotionHandling.Interpreter.GmcIpUserConfig.gmcipus.dob, gmcipuc <- MotionHandling.Interpreter.GmcIpUserConfig.gmcipuc.dob
VcDataObjects: Visu <- Visualization.Visu.dob
Binaries: TRFk_A0, arnc0001, sysconf, asfw, ashwd, arconfig, iomap, acp10cfg, arnc0map, arnc0cfg, acp10map, cncmap, axesmap, Acp10sys, Arnc0sys, Visu102, Visu101, burgf5oe, MP50Ke01, MP50Ke03, MP50Ke02, vccscale, vccpopup, vccddbox, courbd, vccslider, vccdt, Visu01, vccalarm, arialbd, vcchspot, vccshape, vccedit, vccbmp, arialxsr, dejavz0z, vcclbox, vcctext, Visu03, vccbtn, vccstr, vccline, vccovl, Visu02, vccnum, vcpkat, vcpdvnc, vcshared, vcfile, arial, vcpfx20, vcgclass, vcrt, vcfntttf, vcalarm, vcdsint, vctcal, vcmgr, vcdsloc, vcresman, visvc, vcnet, vcpdsw, vcbclass
Libraries: Acp10man, Acp10par, NcGlobal, Runtime, Operator, AsIecCon, astime, DataObj, AsMem, AsArLog, sys_lib, AsArProf, brsystem, FileIO, standard, asrfbext, AsICMP, AsUSB, visapi, TRF_LIB, AsIO, AsIOMMan, AsIODiag, AsSem, Acp10_MC, Acp10sdc, Acp10sim, AsBrStr, ModDiag, MyLib, Arnc0ext, Arnc0man, Arnc0mx, powerlnk, loopconr, ashw
```

### Hardware
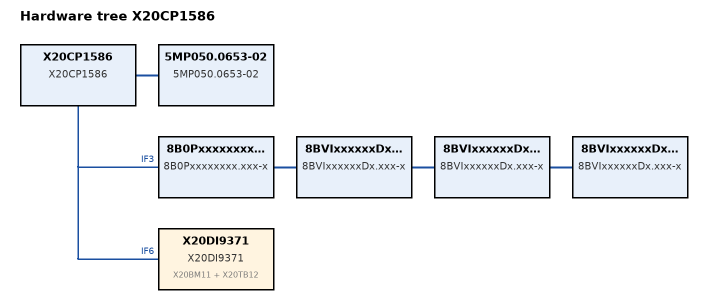
```
5MP050.0653-02 : 5MP050.0653-02 v1.0.3.0  [ETH1 -> X20CP1586.IF2 (NodeNumber=1)]
  Terminal = true
  VncVcObjectName = Visu
  VncKeyMappingFile = VC\5MP050.0653-02.dis
  VncAuthentication = 1
  VncPasswordViewOnly = 1
  VncPasswordViewControl = 2
  VncMaxConnections = 8
  VncRefreshRate = 100
  VncTitle = 6AxesRobot
8B0Pxxxxxxxx.xxx-x : 8B0Pxxxxxxxx.xxx-x v1.0.0.3 (Disabled=true)  [PLK1 -> X20CP1586.IF3 (NodeNumber=1); PLK2 -> 8BVIxxxxxxDx.xxx-x.PLK1 (NodeNumber=1)]
8BVIxxxxxxDx.xxx-x : 8BVIxxxxxxDx.xxx-x v1.0.0.7 (Disabled=true)  [PLK1 -> 8B0Pxxxxxxxx.xxx-x.PLK2 (NodeNumber=2); PLK2 -> 8BVIxxxxxxDx.xxx-x1.PLK1 (NodeNumber=2)]
8BVIxxxxxxDx.xxx-x1 : 8BVIxxxxxxDx.xxx-x v1.0.0.7 (Disabled=true)  [PLK1 -> 8BVIxxxxxxDx.xxx-x.PLK2 (NodeNumber=3); PLK2 -> 8BVIxxxxxxDx.xxx-x2.PLK1 (NodeNumber=3)]
8BVIxxxxxxDx.xxx-x2 : 8BVIxxxxxxDx.xxx-x v1.0.0.7 (Disabled=true)  [PLK1 -> 8BVIxxxxxxDx.xxx-x1.PLK2 (NodeNumber=4)]
X20BM11 : X20BM11 v1.0.0.0 (Disabled=true)  [X2X1 -> X20CP1586.IF6]
X20CP1586 : X20CP1586 v1.0.5.0
  Connector IF2:
    ActivateDevice = 1
    EthInterfaceRedundant = 0
    Mode = Manual
    InternetAddress = 192.168.1.9
    SubnetMask = 255.255.255.0
  Connector IF3:
    EplInterfaceRedundant = 0
    Channel1
    ChannelID1 = ACP10_MC_BROADCAST
    ChannelType1 = OCTET[96]
    EplEthInterfaceRedundant = 0
  UserRamSize = 770048
  RemanentGlobalPvSize = 81920
  VolatileGlobalPvSize = 500000
  BRObjects = 500
  EnableUsbRemoteInstall = 1
  Connections = 8
  TimerDeviceType = EPLX2X
  TimerDevice = X20CP1586.IF3
  TaskClassIdleTime = 4000
  Cyclic1Duration = 4000
  Cyclic1Tolerance = 0
  Cyclic1Stack = 400000
  Cyclic1Output = 1
  Cyclic2Duration = 30000
  Cyclic2Tolerance = 30000
  Cyclic2Stack = 28192
  Cyclic3Duration = 20000
  Cyclic3Tolerance = 30000000
  Cyclic3Stack = 81920
  Cyclic4Duration = 100000
  Cyclic4Tolerance = 100000
  Cyclic5Duration = 200000
  Cyclic5Tolerance = 200000
  Cyclic6Duration = 500000
  Cyclic6Tolerance = 500000
  Cyclic7Duration = 1000000
  Cyclic7Tolerance = 1000000
  Cyclic8Duration = 30000
  Cyclic8Tolerance = 30000000
  Cyclic8Stack = 38192
  FileDevice1
  FileDeviceName1 = CNC_PrgDir
  FileDevicePath1 = C:\Data\Programs
X20DI9371 : X20DI9371 v1.0.1.2 (Disabled=true)  [SS1 -> X20TB12.SS; SL -> X20BM11.SL1]
X20TB12 : X20TB12 v1.0.0.0 (Disabled=true)
```

### IoMap.iom - X20CP1586/IoMap.iom
```iecst
(********************************************************************
 * COPYRIGHT --
 ********************************************************************
 * File: IoMap.iom
 * Author: renj
 * Created: November 11, 2014
 ********************************************************************
 * IO mapping file
 ********************************************************************)
VAR_CONFIG
	DI1.I1 AT %IX."X20DI9371".DigitalInput01;
	DI1.I2 AT %IX."X20DI9371".DigitalInput02;
	DI1.I3 AT %IX."X20DI9371".DigitalInput03;
	DI1.I4 AT %IX."X20DI9371".DigitalInput04;
	DI1.I5 AT %IX."X20DI9371".DigitalInput05;
	DI1.I6 AT %IX."X20DI9371".DigitalInput06;
	DI1.I7 AT %IX."X20DI9371".DigitalInput07;
	DI1.I8 AT %IX."X20DI9371".DigitalInput08;
	DI1.I9 AT %IX."X20DI9371".DigitalInput09;
	DI1.I10 AT %IX."X20DI9371".DigitalInput10;
	DI1.I11 AT %IX."X20DI9371".DigitalInput11;
	DI1.I12 AT %IX."X20DI9371".DigitalInput12;
END_VAR
```

### AXESMap.ncm - X20CP1586/Motion/AXESMap.ncm
```
NcMapping (NcSwId=ACP10, DisabledNodesAreHidden=False)
  NcObject gPowerSupply (ModuleAddress=SDC_IF1.ST7, InterfaceType=SDC, Type=ncAXIS, Channel=1, AcoposSimulation=Off, InitParameter=sdc_i, AcoposParameter=sdc_p, Disabled=FALSE)
  NcObject gAxisQ1 (ModuleAddress=SDC_IF1.ST8, InterfaceType=SDC, Type=ncAXIS, Channel=1, AcoposSimulation=Off, InitParameter=sdc_j1_i, AcoposParameter=sdc_p, AdditionalData=CNC_Enabled="1", Disabled=FALSE)
  NcObject gAxisQ2 (ModuleAddress=SDC_IF1.ST9, InterfaceType=SDC, Type=ncAXIS, Channel=1, AcoposSimulation=Off, InitParameter=sdc_j2_i, AcoposParameter=sdc_p, AdditionalData=CNC_Enabled="1", Disabled=FALSE)
  NcObject gAxisQ3 (ModuleAddress=SDC_IF1.ST10, InterfaceType=SDC, Type=ncAXIS, Channel=1, AcoposSimulation=Off, InitParameter=sdc_j3_i, AcoposParameter=sdc_p, AdditionalData=CNC_Enabled="1", Disabled=FALSE)
  NcObject gAxisQ4 (ModuleAddress=SDC_IF1.ST11, InterfaceType=SDC, Type=ncAXIS, Channel=1, AcoposSimulation=Off, InitParameter=sdc_j4_i, AcoposParameter=sdc_p, AdditionalData=CNC_Enabled="1", Disabled=FALSE)
  NcObject gAxisQ5 (ModuleAddress=SDC_IF1.ST12, InterfaceType=SDC, Type=ncAXIS, Channel=1, AcoposSimulation=Off, InitParameter=sdc_j5_i, AcoposParameter=sdc_p, AdditionalData=CNC_Enabled="1", Disabled=FALSE)
  NcObject gAxisQ6 (ModuleAddress=SDC_IF1.ST13, InterfaceType=SDC, Type=ncAXIS, Channel=1, AcoposSimulation=Off, InitParameter=sdc_j6_i, AcoposParameter=sdc_p, AdditionalData=CNC_Enabled="1", Disabled=FALSE)
  NcObject gAxisX (ModuleAddress=SDC_IF1.ST1, InterfaceType=SDC, Type=ncAXIS, Channel=1, AcoposSimulation=Off, InitParameter=sdc_i, AcoposParameter=sdc_p, AdditionalData=CNC_Enabled="1", Disabled=FALSE, ModuleDisabled=FALSE)
  NcObject gAxisY (ModuleAddress=SDC_IF1.ST2, InterfaceType=SDC, Type=ncAXIS, Channel=1, AcoposSimulation=Off, InitParameter=sdc_i, AcoposParameter=sdc_p, AdditionalData=CNC_Enabled="1", Disabled=FALSE)
  NcObject gAxisZ (ModuleAddress=SDC_IF1.ST3, InterfaceType=SDC, Type=ncAXIS, Channel=1, AcoposSimulation=Off, InitParameter=sdc_i, AcoposParameter=sdc_p, AdditionalData=CNC_Enabled="1", Disabled=FALSE)
  NcObject gAxisA (ModuleAddress=SDC_IF1.ST4, InterfaceType=SDC, Type=ncAXIS, Channel=1, AcoposSimulation=Off, InitParameter=sdc_i, AcoposParameter=sdc_p, AdditionalData=CNC_Enabled="1", Disabled=FALSE)
  NcObject gAxisB (ModuleAddress=SDC_IF1.ST5, InterfaceType=SDC, Type=ncAXIS, Channel=1, AcoposSimulation=Off, InitParameter=sdc_i, AcoposParameter=sdc_p, AdditionalData=CNC_Enabled="1", Disabled=FALSE)
  NcObject gAxisC (ModuleAddress=SDC_IF1.ST6, InterfaceType=SDC, Type=ncAXIS, Channel=1, AcoposSimulation=Off, InitParameter=sdc_i, AcoposParameter=sdc_p, AdditionalData=CNC_Enabled="1", Disabled=FALSE)
```

### Acp10cfg.ncc - X20CP1586/Motion/Acp10cfg.ncc
```
NcConfiguration (Version=2.46.0, NcSwId=Acp10)
  ACP10CF1_typ:
    cnt_nettrc_rec_drive = 1500
    bufsize_trace_upload = 1200
    tc_nc_man_task = Cyclic #1
    glob_pv_as_ncobject = Yes
    ncsys_dl_broadcast = Yes
    ncsys_dl_acp_reset = Yes
    safemc_log_err_to_ax = Yes
    network_init:
      ncsw_init_execute = Yes
      automatic_execute = No
      node_nr_warning = Yes
      net_err_before_ncact = Yes
    nettrc:
      enter_parsecrec = Yes
      enter_ncaction = Yes
      save_ring_startidx = Yes
    cam_prof_download:
      cam_dat_dl_parallel = No
      tc_cam_dl_parallel = Task class for NC Manager task
    plk_if[0]:
      if_name = IF3
      tc_CycDat_PLCopen = Task class for NC Manager task
      mc_broadcast_extdat = No
    sdc_if[0]:
      if_name = SDC_IF1
      mc_broadcast_size = 800
      mc_broadcast_extdat = No
```

### Acp10map.ncm - X20CP1586/Motion/Acp10map.ncm
```
NcMapping (NcSwId=Acp10, DisabledNodesAreHidden=False)
  NcObject 8B0Pxxxxxxxx.xxx-x_ncAXIS2 (ModuleId=8B0Pxxxxxxxx.xxx-x, Type=ncAXIS, Channel=2, AcoposSimulation=Off, Disabled=TRUE, ModuleDisabled=FALSE)
  NcObject 8B0Pxxxxxxxx.xxx-x_ncV_AXIS1 (ModuleId=8B0Pxxxxxxxx.xxx-x, Type=ncV_AXIS, Channel=1, Disabled=TRUE, ModuleDisabled=FALSE)
  NcObject 8B0Pxxxxxxxx.xxx-x_ncV_AXIS2 (ModuleId=8B0Pxxxxxxxx.xxx-x, Type=ncV_AXIS, Channel=2, Disabled=TRUE, ModuleDisabled=FALSE)
  NcObject 8BVIxxxxxxDx.xxx-x_ncV_AXIS1 (ModuleId=8BVIxxxxxxDx.xxx-x, Type=ncV_AXIS, Channel=1, Disabled=TRUE, ModuleDisabled=FALSE)
  NcObject 8BVIxxxxxxDx.xxx-x_ncV_AXIS2 (ModuleId=8BVIxxxxxxDx.xxx-x, Type=ncV_AXIS, Channel=2, Disabled=TRUE, ModuleDisabled=FALSE)
  NcObject 8BVIxxxxxxDx.xxx-x1_ncV_AXIS1 (ModuleId=8BVIxxxxxxDx.xxx-x1, Type=ncV_AXIS, Channel=1, Disabled=TRUE, ModuleDisabled=FALSE)
  NcObject 8BVIxxxxxxDx.xxx-x1_ncV_AXIS2 (ModuleId=8BVIxxxxxxDx.xxx-x1, Type=ncV_AXIS, Channel=2, AcoposParameter=acpmic_p, Disabled=TRUE, ModuleDisabled=FALSE)
  NcObject 8BVIxxxxxxDx.xxx-x2_ncV_AXIS1 (ModuleId=8BVIxxxxxxDx.xxx-x2, Type=ncV_AXIS, Channel=1, Disabled=TRUE, ModuleDisabled=FALSE)
  NcObject 8BVIxxxxxxDx.xxx-x2_ncV_AXIS2 (ModuleId=8BVIxxxxxxDx.xxx-x2, Type=ncV_AXIS, Channel=2, Disabled=TRUE, ModuleDisabled=FALSE)
  NcObject gPowerSupply (ModuleId=8B0Pxxxxxxxx.xxx-x, Type=ncAXIS, Channel=1, AcoposSimulation=Off, InitParameter=sdc_i, Disabled=TRUE, ModuleDisabled=FALSE)
  NcObject gAxisQ1 (ModuleId=8BVIxxxxxxDx.xxx-x, Type=ncAXIS, Channel=1, AcoposSimulation=Off, InitParameter=joint1_i, AcoposParameter=acpm_p, AdditionalData=CNC_Enabled="1", Disabled=TRUE, ModuleDisabled=FALSE)
  NcObject gAxisQ2 (ModuleId=8BVIxxxxxxDx.xxx-x, Type=ncAXIS, Channel=2, AcoposSimulation=Off, InitParameter=joint2_i, AcoposParameter=acpm_p, AdditionalData=CNC_Enabled="1", Disabled=TRUE, ModuleDisabled=FALSE)
  NcObject gAxisQ3 (ModuleId=8BVIxxxxxxDx.xxx-x1, Type=ncAXIS, Channel=1, AcoposSimulation=Off, InitParameter=joint3_i, AcoposParameter=acpmic_p, AdditionalData=CNC_Enabled="1", Disabled=TRUE, ModuleDisabled=FALSE)
  NcObject gAxisQ4 (ModuleId=8BVIxxxxxxDx.xxx-x1, Type=ncAXIS, Channel=2, AcoposSimulation=Off, InitParameter=joint4_i, AcoposParameter=acpmic_p, AdditionalData=CNC_Enabled="1", Disabled=TRUE, ModuleDisabled=FALSE)
  NcObject gAxisQ5 (ModuleId=8BVIxxxxxxDx.xxx-x2, Type=ncAXIS, Channel=1, AcoposSimulation=Off, InitParameter=joint5_i, AcoposParameter=acpmic_p, AdditionalData=CNC_Enabled="1", Disabled=TRUE, ModuleDisabled=FALSE)
  NcObject gAxisQ6 (ModuleId=8BVIxxxxxxDx.xxx-x2, Type=ncAXIS, Channel=2, AcoposSimulation=Off, InitParameter=joint6_i, AcoposParameter=acpmic_p, AdditionalData=CNC_Enabled="1", Disabled=TRUE, ModuleDisabled=FALSE)
```

### Arnc0cfg.ncc - X20CP1586/Motion/Arnc0cfg.ncc
```
NcConfiguration (Version=1.46.0, NcSwId=Arnc0)
  ARNC0CFG_typ:
    sampling_rate = 2000
    cnt_nettrc_rec_drive = 1500
    bufsize_sys_trace = 16#00005000
    enable_mp_log = Yes
    tc_nc_man_task = Cyclic #1
    bg_load = 1
    glob_pv_as_ncobject = Yes
```

### CNCMap.ncm - X20CP1586/Motion/CNCMap.ncm
```
NcMapping (NcSwId=ARNC0, DisabledNodesAreHidden=False)
  NcObject gRobot (Type=ncCNCSYS, Channel=1, AcoposSimulation=Off, InitParameter=robot_i, Disabled=FALSE, ModuleDisabled=FALSE)
```

## Configuration X20CP3586

CPU , AutomationRuntime V4.04, Build 4.1.2, Safety 1.5

### Task classes (Cpu.sw)
```
Cyclic#1 (cycle 2000 us, tolerance 0 us):
  6axATrqFF <- MotionHandling.FeedForward.6axATrqFF.prg
  Config <- MotionHandling.Configuration.Config.prg
  System <- MotionHandling.SystemHandling.System.prg
  Cnc <- MotionHandling.CncHandling.Cnc.prg
  Axes <- MotionHandling.AxesHandling.Axes.prg
  OptMotion <- MotionHandling.Optimizer.OptMotion.prg
  Jog <- MotionHandling.Jogging.Jog.prg
  Trf <- MotionHandling.Transformations.Trf.prg
Cyclic#2 (cycle 30000 us, tolerance 60000 us):
  Error <- ErrorHandling.Error.prg
  HmiKeyCtrl <- HmiHandling.HmiKeyCtrl.HmiKeyCtrl.prg
  HmiHardKey <- HmiHandling.HmiHardKey.HmiHardKeyCtrl.prg
Cyclic#4 (cycle 100000 us, tolerance 100000 us):
  HmiJogCtrl <- HmiHandling.HmiJog.HmiJogCtrl.prg
  HmiSetup <- HmiHandling.HmiSetup.HmiSetup.prg
Cyclic#8 (cycle 30000 us, tolerance 30000000 us):
  RecipeCont <- Recipe.RecipeControl.prg
  HmiIO <- HmiHandling.HmiIO.HmiIO.prg
  HmiAlarm <- HmiHandling.HmiAlarm.HmiAlarm.prg
DataObjects: Acp10sys, Arnc0sys, acp10sys, arnc0sys, User
NcDataObjects: sdc_i <- MotionHandling.MotionInitFiles.SDC.sdc_i.dob, sdc_p <- MotionHandling.MotionInitFiles.SDC.sdc_p.dob, ps_p <- MotionHandling.MotionInitFiles.ps_p.dob, acpm_p <- MotionHandling.MotionInitFiles.acpm_p.dob, acpmic_p <- MotionHandling.MotionInitFiles.acpmic_p.dob, joint1_i <- MotionHandling.MotionInitFiles.joint1_i.dob, joint2_i <- MotionHandling.MotionInitFiles.joint2_i.dob, joint3_i <- MotionHandling.MotionInitFiles.joint3_i.dob, joint4_i <- MotionHandling.MotionInitFiles.joint4_i.dob, joint5_i <- MotionHandling.MotionInitFiles.joint5_i.dob, joint6_i <- MotionHandling.MotionInitFiles.joint6_i.dob, AcpError <- MotionHandling.AxesHandling.AcpError.dob, JogInit <- MotionHandling.Jogging.JogInit.dob, JogPrg <- MotionHandling.Jogging.JogPrg.dob, robot_i <- MotionHandling.MotionInitFiles.robot_i.dob
Binaries: TRFk_A0, sysconf, ashwd, iomap, asfw, arconfig, acp10cfg, arnc0cfg, cncmap, axesmap, Arnc0map, Acp10map, Acp10sys, Arnc0sys, vcfntttf, vccedit, vccbmp, vcshared, vcpdvnc, vccshape, vcfile, vcgclass, vcchspot, Vismp02, vcmgr, vcresman, vccbtn, vcdsloc, vccalarm, vccovl, vcpfx20, vccline, vcctext, vcalarm, vcbclass, visvc, vcrt, vccnum, vccstr, vcnet, arialbd, Vismp01, vcpdsw, Vismp03, vcdsint, vctcal, vcclbox, vccdt, arial, vccbar, vccddbox, vccpopup, arialxsr, AXESMap, CNCMap, Arnc0cfg, Acp10cfg, Visu03, Visu01, Visu02, arialgkb
Libraries: Operator, AsIecCon, astime, DataObj, AsMem, AsArLog, AsArProf, FileIO, standard, Acp10sim, acp10_mc, brsystem, Acp10man, sys_lib, Runtime, NcGlobal, Acp10par, Acp10sdc, asrfbext, AsICMP, AsUSB, visapi, ModDiag, AsIOMMan, AsIODiag, AsSem, TRF_LIB, AsIO, AsBrStr, powerlnk, MyLib, Arnc0ext, Arnc0man, Arnc0mx, loopconr, ashw
```

### Hardware
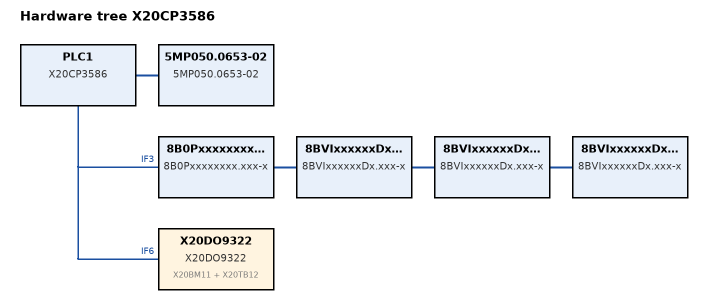
```
5MP050.0653-02 : 5MP050.0653-02 v1.0.3.1  [ETH1 -> PLC1.IF2 (NodeNumber=1)]
  Terminal = true
  VncVcObjectName = Visu
  VncKeyMappingFile = 5MP050.0653-02.dis
  VncAuthentication = 1
  VncPasswordViewOnly = 1
  VncPasswordViewControl = 2
8B0Pxxxxxxxx.xxx-x : 8B0Pxxxxxxxx.xxx-x v1.0.0.3 (Disabled=true)  [PLK1 -> PLC1.IF3 (NodeNumber=1); PLK2 -> 8BVIxxxxxxDx.xxx-x.PLK1 (NodeNumber=1)]
  OrderNumber = 8B0P0220HW00.000-1
8BVIxxxxxxDx.xxx-x : 8BVIxxxxxxDx.xxx-x v1.0.0.7 (Disabled=true)  [PLK1 -> 8B0Pxxxxxxxx.xxx-x.PLK2 (NodeNumber=2); PLK2 -> 8BVIxxxxxxDx.xxx-x1.PLK1 (NodeNumber=2)]
8BVIxxxxxxDx.xxx-x1 : 8BVIxxxxxxDx.xxx-x v1.0.0.7 (Disabled=true)  [PLK1 -> 8BVIxxxxxxDx.xxx-x.PLK2 (NodeNumber=3); PLK2 -> 8BVIxxxxxxDx.xxx-x2.PLK1 (NodeNumber=3)]
8BVIxxxxxxDx.xxx-x2 : 8BVIxxxxxxDx.xxx-x v1.0.0.7 (Disabled=true)  [PLK1 -> 8BVIxxxxxxDx.xxx-x1.PLK2 (NodeNumber=4)]
PLC1 : X20CP3586 v1.0.5.0
  Connector IF2:
    ActivateDevice = 1
    EthInterfaceRedundant = 0
    Mode = Manual
    InternetAddress = 192.168.1.9
    SubnetMask = 255.255.255.0
    Vnc1
    VncVcObjectName1 = Visu
    VncKeyMappingFile1 = VC\PS2-Keyboard.dis
    VncAuthentication1 = 1
    VncPasswordViewOnly1 = v
    VncPasswordViewControl1 = c
    VncPortNumber1 = 5901
    VncRefreshRate1 = 100
    Vnc2
    VncVcObjectName2 = MP50Ke
    VncKeyMappingFile2 = VC\PS2-Keyboard1.dis
    VncAuthentication2 = 1
    VncPasswordViewOnly2 = v
    VncPasswordViewControl2 = c
    VncPortNumber2 = 5902
    VncRefreshRate2 = 100
  Connector IF3:
    EplInterfaceRedundant = 0
    Channel1
    ChannelID1 = ACP10_MC_BROADCAST
    ChannelType1 = OCTET[48]
    EplEthInterfaceRedundant = 0
  UserRamSize = 770048
  RemanentGlobalPvSize = 81920
  VolatileGlobalPvSize = 500000
  EnableUsbRemoteInstall = 1
  Connections = 8
  TimerDeviceType = EPLX2X
  TimerDevice = PLC1.IF3
  TaskClassIdleTime = 8000
  Cyclic1Duration = 2000
  Cyclic1Tolerance = 0
  Cyclic1Stack = 40000
  Cyclic1Output = 1
  Cyclic2Duration = 30000
  Cyclic2Tolerance = 60000
  Cyclic2Stack = 28192
  Cyclic3Duration = 50000
  Cyclic3Tolerance = 200000
  Cyclic3Stack = 10240
  Cyclic4Duration = 100000
  Cyclic4Tolerance = 100000
  Cyclic5Duration = 200000
  Cyclic5Tolerance = 200000
  Cyclic6Duration = 500000
  Cyclic6Tolerance = 500000
  Cyclic7Duration = 1000000
  Cyclic7Tolerance = 1000000
  Cyclic8Duration = 30000
  Cyclic8Tolerance = 30000000
  Cyclic8Stack = 38192
  FileDevice1
  FileDeviceName1 = CNC_PrgDir
  FileDevicePath1 = C:\Data\Programs
X20BM11 : X20BM11 v1.0.0.0 (Disabled=true)  [X2X1 -> PLC1.IF6]
X20DO9322 : X20DO9322 v1.0.2.2 (Disabled=true)  [SS1 -> X20TB12i.SS; SL -> X20BM11.SL1]
X20TB12i : X20TB12 v1.0.0.0 (Disabled=true)
```

### AXESMap.ncm - PLC1/Motion/AXESMap.ncm
```
NcMapping (NcSwId=ACP10)
  NcObject gAxisX (ModuleAddress=SDC_IF1.ST1, InterfaceType=SDC, Type=ncAXIS, Channel=1, AcoposSimulation=Off, InitParameter=sdc_i, AcoposParameter=sdc_p, AdditionalData=CNC_Enabled="1", Disabled=FALSE, ModuleDisabled=FALSE)
  NcObject gAxisY (ModuleAddress=SDC_IF1.ST2, InterfaceType=SDC, Type=ncAXIS, Channel=1, AcoposSimulation=Off, InitParameter=sdc_i, AcoposParameter=sdc_p, AdditionalData=CNC_Enabled="1", Disabled=FALSE)
  NcObject gAxisZ (ModuleAddress=SDC_IF1.ST3, InterfaceType=SDC, Type=ncAXIS, Channel=1, AcoposSimulation=Off, InitParameter=sdc_i, AcoposParameter=sdc_p, AdditionalData=CNC_Enabled="1", Disabled=FALSE)
  NcObject gAxisA (ModuleAddress=SDC_IF1.ST4, InterfaceType=SDC, Type=ncAXIS, Channel=1, AcoposSimulation=Off, InitParameter=sdc_i, AcoposParameter=sdc_p, AdditionalData=CNC_Enabled="1", Disabled=FALSE)
  NcObject gAxisB (ModuleAddress=SDC_IF1.ST5, InterfaceType=SDC, Type=ncAXIS, Channel=1, AcoposSimulation=Off, InitParameter=sdc_i, AcoposParameter=sdc_p, AdditionalData=CNC_Enabled="1", Disabled=FALSE)
  NcObject gAxisC (ModuleAddress=SDC_IF1.ST6, InterfaceType=SDC, Type=ncAXIS, Channel=1, AcoposSimulation=Off, InitParameter=sdc_i, AcoposParameter=sdc_p, AdditionalData=CNC_Enabled="1", Disabled=FALSE)
```

### Acp10cfg.ncc - PLC1/Motion/Acp10cfg.ncc
```
NcConfiguration (Version=2.37.0, NcSwId=acp10)
  ACP10CF1_typ:
    cnt_nettrc_rec_drive = 1500
    bufsize_trace_upload = 1200
    tc_nc_man_task = Cyclic #1
    glob_pv_as_ncobject = Yes
    ncsys_dl_broadcast = Yes
    ncsys_dl_acp_reset = Yes
    network_init:
      ncsw_init_execute = Yes
      automatic_execute = No
      node_nr_warning = Yes
      net_err_before_ncact = Yes
    nettrc:
      enter_parsecrec = Yes
      enter_ncaction = Yes
      save_ring_startidx = Yes
    plk_if[0]:
      if_name = IF3
      tc_CycDat_PLCopen = Task class for NC Manager task
      mc_broadcast_extdat = No
    sdc_if[0]:
      if_name = SDC_IF1
      mc_broadcast_size = 800
      mc_broadcast_extdat = No
```

### Acp10map.ncm - PLC1/Motion/Acp10map.ncm
```
NcMapping (NcSwId=Acp10)
  NcObject gPowerSupply (ModuleId=8B0Pxxxxxxxx.xxx-x, Type=ncAXIS, Channel=1, AcoposSimulation=Off, InitParameter=sdc_i, Disabled=FALSE, ModuleDisabled=FALSE)
  NcObject gAxisQ1 (ModuleId=8BVIxxxxxxDx.xxx-x, Type=ncAXIS, Channel=1, AcoposSimulation=Off, InitParameter=joint1_i, AcoposParameter=acpm_p, AdditionalData=CNC_Enabled="1", Disabled=FALSE, ModuleDisabled=FALSE)
  NcObject gAxisQ2 (ModuleId=8BVIxxxxxxDx.xxx-x, Type=ncAXIS, Channel=2, AcoposSimulation=Off, InitParameter=joint2_i, AcoposParameter=acpm_p, AdditionalData=CNC_Enabled="1", Disabled=FALSE, ModuleDisabled=FALSE)
  NcObject gAxisQ3 (ModuleId=8BVIxxxxxxDx.xxx-x1, Type=ncAXIS, Channel=1, AcoposSimulation=Off, InitParameter=joint3_i, AcoposParameter=acpmic_p, AdditionalData=CNC_Enabled="1", Disabled=FALSE, ModuleDisabled=FALSE)
  NcObject gAxisQ4 (ModuleId=8BVIxxxxxxDx.xxx-x1, Type=ncAXIS, Channel=2, AcoposSimulation=Off, InitParameter=joint4_i, AcoposParameter=acpmic_p, AdditionalData=CNC_Enabled="1", Disabled=FALSE, ModuleDisabled=FALSE)
  NcObject gAxisQ5 (ModuleId=8BVIxxxxxxDx.xxx-x2, Type=ncAXIS, Channel=1, AcoposSimulation=Off, InitParameter=joint5_i, AcoposParameter=acpmic_p, AdditionalData=CNC_Enabled="1", Disabled=FALSE, ModuleDisabled=FALSE)
  NcObject gAxisQ6 (ModuleId=8BVIxxxxxxDx.xxx-x2, Type=ncAXIS, Channel=2, AcoposSimulation=Off, InitParameter=joint6_i, AcoposParameter=acpmic_p, AdditionalData=CNC_Enabled="1", Disabled=FALSE, ModuleDisabled=FALSE)
```

### CNCMap.ncm - PLC1/Motion/CNCMap.ncm
```
NcMapping (NcSwId=ARNC0)
  NcObject gRobot (ModuleAddress=ST1, Type=ncCNCSYS, Channel=1, AcoposSimulation=Off, InitParameter=cnc_i, Disabled=FALSE, ModuleDisabled=FALSE)
```

## Logical view

Binary libraries used (declarations not repeated): Runtime, Operator, AsIecCon, astime, DataObj, AsMem, AsArLog, sys_lib, AsArProf, brsystem, FileIO, standard, asrfbext, AsICMP, AsUSB, visapi, TRF_LIB 2.02.0, AsIO, AsIOMMan, AsIODiag, AsSem, AsBrStr, Arnc0ext 2.47.4, LoopConR 2.80.9, Acp10man 2.48.1, Acp10par 2.48.1, NcGlobal 2.48.1, Acp10sim 2.48.1, Acp10_MC 2.48.1, Arnc0man 2.48.1, Acp10sdc 2.48.1, Arnc0mx 2.48.1

### Global.var - Axes Definition
```iecst
(********************************************************************
 * COPYRIGHT -- Bernecker + Rainer
 ********************************************************************
 * File: Global.var
 * Author: frigenif
 * Created: December 05, 2012
 ********************************************************************
 * Global variables of project Estun
 ********************************************************************)
VAR
	gAxisQ1 : ACP10AXIS_typ := (0);
	gAxisQ2 : ACP10AXIS_typ := (0);
	gAxisQ3 : ACP10AXIS_typ := (0);
	gAxisQ4 : ACP10AXIS_typ := (0);
	gAxisQ5 : ACP10AXIS_typ := (0);
	gAxisQ6 : ACP10AXIS_typ := (0);
	gAxisX : ACP10AXIS_typ := (0);
	gAxisY : ACP10AXIS_typ := (0);
	gAxisZ : ACP10AXIS_typ := (0);
	gAxisA : ACP10AXIS_typ := (0);
	gAxisB : ACP10AXIS_typ := (0);
	gAxisC : ACP10AXIS_typ := (0);
	gPowerSupply : ACP10AXIS_typ := (0);
	gAxisFrameX : ACP10AXIS_typ := (0);
	gRobot : ARNC0CNC_typ := (0);
END_VAR
```

### Package Logical/Libraries - Global libraries

### Library Logical/Libraries/MyLib (ANSIC) - Including Stringhelper and ST Handler
